FUNCTION_BLOCK FB_TemperatureAfterGearbox
VAR_INPUT
	TemperatureBeforeGearbox : REAL ; // Celcius
	PumpFlow : REAL ; // L/s
	Density : REAL ; // g/L
	SpecificHeatCapacity : REAL ; //  j/(g C) 
	GearboxEfficiency : REAL ; //%, 0-1
	Gearboxheat : REAL ; // Watt
	GearboxStandardHeat : REAL ; // Watt
	TotalPipeVolume : REAL ; // L
	CurrentPipeVolume : REAL ; // L
	BoolSimulationTesting : BOOL ;
END_VAR
VAR_OUTPUT
	TemperatureAfterGearbox : REAL := Simulation_Parameters.AmbientTemperature ; // L
END_VAR
VAR
	SurgeValvePosition : REAL ; // % 0-1
	deltaTByGearboxHeat : REAL ; // Celsius
	deltaTByGearboxStandardHeat : REAL ; // Celsius
	deltaTByGearboxHeatEfficiencyCorrected : REAL ; // Celsius
	
	MimimumPipeVolumeForHeatTransfer : REAL ; // L
	TemperatureAfterGearboxNonFiltered : REAL ; // Celsius
END_VAR

IF NOT BoolSimulationTesting THEN
	SurgeValvePosition := 0.05; //Use hardcoded SurgeValvePosition
ELSE
	; //Frank Logic for SurgeValvePosition.
END_IF


MimimumPipeVolumeForHeatTransfer := TotalPipeVolume*3/4;

IF CurrentPipeVolume <= MimimumPipeVolumeForHeatTransfer THEN
	deltaTByGearboxHeat := 0 ;
	deltaTByGearboxStandardHeat := 0 ;
	
ELSE 
	deltaTByGearboxHeat := f_CalculateDeltaT(SpecificHeatCapacity := SpecificHeatCapacity,
											Density := Density,
											Mass := PumpFlow,
											PowerInput := Gearboxheat);
								
	deltaTByGearboxStandardHeat := f_CalculateDeltaT(SpecificHeatCapacity := SpecificHeatCapacity,
													Density := Density,
													Mass := PumpFlow,
													PowerInput := GearboxStandardHeat); 
	deltaTByGearboxHeatEfficiencyCorrected := (1-GearboxEfficiency) * deltaTByGearboxHeat;
						
	TemperatureAfterGearboxNonFiltered := TemperatureBeforeGearbox + (SurgeValvePosition *  deltaTByGearboxHeatEfficiencyCorrected) + deltaTByGearboxStandardHeat;
	TemperatureAfterGearbox := (1-simulation_parameters.TimeConstantGearbox)*TemperatureAfterGearbox + simulation_parameters.TimeConstantGearbox*TemperatureAfterGearboxNonFiltered ;

END_IF

END_FUNCTION_BLOCK

(* stored: Version 1.1.0.1, ProductVersion 3.1.4024.12
   POU FB_TemperatureAfterGearbox: Id {26c4ff50-fec5-40fc-8b57-ba9d53fbda82}, SpecialFunc None *)
